// provide API method calls to retreive IO status, Recipe Management Status and controller status.
FUNCTION_BLOCK T_Data
VAR_INPUT
END_VAR
VAR_OUTPUT
END_VAR
VAR
END_VAR

{attribute 'TcRpcEnable'}
METHOD PUBLIC GetIO : ST_IO_Status
VAR_INST
    cnt : INT;
END_VAR
GetIO := IO.IO_Status;
cnt := cnt + 1;
END_METHOD

{attribute 'TcRpcEnable'}
METHOD PUBLIC GetIOAsJson : JsonDoc
VAR_INST
    cnt : INT;
END_VAR
VAR 
	jsonDocToProp : FB_JsonReadWriteDatatype;
	sizeOfJDoc : UDINT;
END_VAR
VAR_INST
	sizeOfDoc : UDINT;
	jDoc : JsonDoc;
END_VAR
sizeOfDoc := SIZEOF(jDoc);
jsonDocToProp.GetJsonFromSymbol('ST_IO_Status',SIZEOF(IO.IO_Status), ADR(IO.IO_Status), sizeOfDoc, ADR(jDoc));
GetIOAsJson := jDoc;
cnt := cnt + 1;
END_METHOD

{attribute 'TcRpcEnable'}
METHOD PUBLIC SetIOAsJson : UDINT;
VAR_INPUT
	jDocIn : JsonDoc;
END_VAR
VAR_OUTPUT
	
END_VAR
VAR_INST
    cnt : INT;
END_VAR
VAR 
	jsonDocToProp : FB_JsonReadWriteDatatype;
	sizeOfJDoc : UDINT;
END_VAR
VAR_INST
	sizeOfDoc : UDINT;
	jDoc : JsonDoc;
	localIO : ST_IO_Status;
END_VAR
SetIOAsJson := SIZEOF(jDocIn);
jDoc := jDocIn;
jsonDocToProp.SetSymbolFromJson( jDocIn, 'ST_IO_Status',SIZEOF(localIo), ADR(localIo));
cnt := cnt + 1;
END_METHOD

END_FUNCTION_BLOCK

(* stored: Version 1.1.0.1, ProductVersion 3.1.4024.9
   POU T_Data: Id {f5274923-7677-4878-8f42-4f7d00aba597}, SpecialFunc None
   Method GetIO: Id {ec4027c0-e26b-48ab-b95c-2e5556ef48aa}
   Method GetIOAsJson: Id {e5726361-c4a6-49cc-8229-ef38a2fa04ec}
   Method SetIOAsJson: Id {ae2f91ce-d980-4f4a-814c-1278bb2be93a} *)
